FUNCTION_BLOCK EL3124
VAR
	_io : EL3xx4_Data;
	{attribute addProperty Name "WcState"}
	_wcState : WcStateInputToggle;
	{attribute addProperty Name "Info data"}
	_infoData : InfoDataAds;
END_VAR

PROPERTY IO : REFERENCE TO EL3xx4_Data
GET
IO REF= _io;
END_GET
END_PROPERTY

PROPERTY WcState : REFERENCE TO WcStateInputToggle
GET
WcState REF= _wcState;
END_GET
END_PROPERTY

END_FUNCTION_BLOCK

(* stored: Version 1.1.0.1, ProductVersion 3.1.4024.9
   POU EL3124: Id {1150d13a-f44d-06d4-088a-8031fb5e488f}, SpecialFunc None
   Property IO: Id {4ad6815d-d3fe-0709-1522-f029e7227680}
   Get Get: Id {1390db82-05e4-02f3-243b-94f93ee079af}
   Property WcState: Id {fe9d0c73-ade9-0359-19de-d7aa031d682a}
   Get Get: Id {75e3bcbf-ccdf-07a2-01ca-d795a7099ea5} *)
